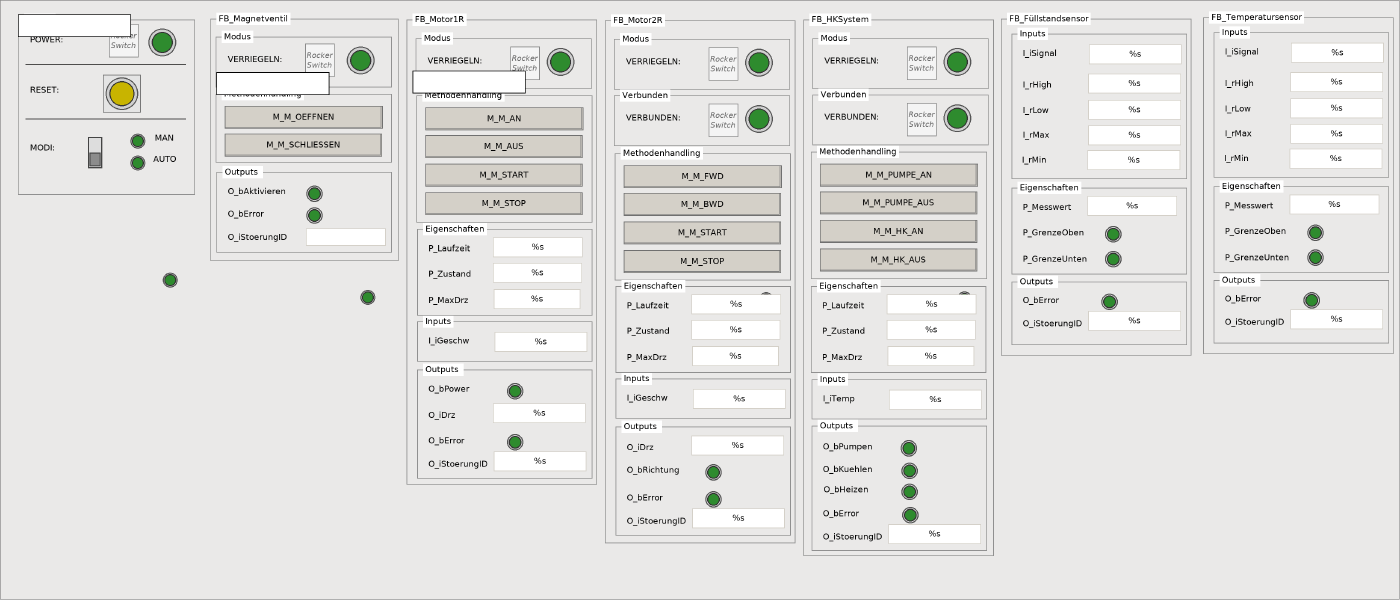
VISUALIZATION Aktoren  // 1863x799
    Rectangle (-1,-1 1863x799)
    GroupBox (280,17 250x330), "FB_Magnetventil"
        Textfield (127,287 106x23), text variable: Reaktoranlage.VENTIL.O_iStoerungID
    GroupBox (287,41 234x75), "Modus"
        Label (13,23 150x30), "VERRIEGELN:"
        Lamp1 (172,18 42x43), variable: Reaktoranlage.VENTIL.I_bVerriegeln, style: Lamp-Lamp1-Green
        Lamp1 (191,340 23x30), style: Lamp-Lamp1-Green
    RockerSwitch (406,58 39x44), variable: Reaktoranlage.VENTIL.I_bVerriegeln, behaviour: TOGGLE, style: Switch-RockerSwitch-Gray
    GroupBox (287,117 234x99), "Methodenhandling"
        Rectangle (-530,-100 150x30)
        Button (12,24 210x30), "M_M_OEFFNEN"
            OnMouseClick: execute { Reaktoranlage.VENTIL.M_M_OEFFNEN(); }
        Button (12,61 209x30), "M_M_SCHLIESSEN"
            OnMouseClick: execute { Reaktoranlage.VENTIL.M_M_SCHLIESSEN(); }
    GroupBox (288,221 233x115), "Outputs"
        Label (12,19 150x30), "O_bAktivieren"
        Label (12,49 150x30), "O_bError"
        Label (12,80 150x30), "O_iStoerungID"
        Lamp1 (118,22 25x30), variable: Reaktoranlage.VENTIL.O_bAktivieren, style: Lamp-Lamp1-Green
        Lamp1 (118,51 25x30), variable: Reaktoranlage.VENTIL.O_bStoerung, style: Lamp-Lamp1-Green
    GroupBox (24,18 235x241), "Modus"
        Label (13,20 150x30), "POWER:"
        RockerSwitch (121,14 39x44), variable: Reaktoranlage.Modus.I_bPower, behaviour: TOGGLE, style: Switch-RockerSwitch-Gray
        Label (13,164 150x30), "MODI:"
        DipSwitch (82,161 41x48), variable: Reaktoranlage.Modus.I_bMode, behaviour: TOGGLE, style: Switch-DipSwitch-Gray
        Lamp1 (148,155 23x30), variable: Reaktoranlage.Modus.O_bMAN, style: Lamp-Lamp1-Green
        Lamp1 (148,184 23x30), variable: Reaktoranlage.Modus.O_bAUTO, style: Lamp-Lamp1-Green
        Label (177,179 46x30), "AUTO"
        Lamp1 (191,340 23x30), style: Lamp-Lamp1-Green
        Line (10,67) (223,67)
        Lamp1 (171,17 42x43), variable: Reaktoranlage.Modus.I_bPower, style: Lamp-Lamp1-Green
        Label (179,151 46x30), "MAN"
        Label (13,87 150x30), "RESET:"
        PushSwitch (113,80 50x53), variable: GVL.VIS_SysReset, behaviour: TAP, style: Switch-PushSwitch-Yellow
        Line (10,140) (223,140)
    GroupBox (541,18 253x627), "FB_Motor1R"
        GroupBox (12,25 234x75), "Modus"
            Label (13,23 150x30), "VERRIEGELN:"
            Lamp1 (172,18 42x43), variable: Reaktoranlage.RUEHRER.I_bVerriegeln, style: Lamp-Lamp1-Green
            Lamp1 (191,340 23x30), style: Lamp-Lamp1-Green
            RockerSwitch (126,19 39x44), variable: Reaktoranlage.RUEHRER.I_bVerriegeln, behaviour: TOGGLE, style: Switch-RockerSwitch-Gray
        GroupBox (13,101 234x177), "Methodenhandling"
            Rectangle (-530,-100 150x30)
            Button (12,24 210x30), "M_M_AN"
                OnMouseClick: execute { Reaktoranlage.RUEHRER.M_M_AN(); }
            Button (12,61 209x30), "M_M_AUS"
                OnMouseClick: execute { Reaktoranlage.RUEHRER.M_M_AUS(); }
            Button (12,99 209x30), "M_M_START"
                OnMouseClick: execute { Reaktoranlage.RUEHRER.M_M_START(); }
            Button (12,137 209x30), "M_M_STOP"
                OnMouseClick: execute { Reaktoranlage.RUEHRER.M_M_STOP(); }
        GroupBox (14,402 233x61), "Inputs"
            Label (12,19 150x30), "I_iGeschw"
            Textfield (103,22 123x26), "%s", text variable: Reaktoranlage.RUEHRER.I_iGeschw
                OnMouseClick: write Reaktoranlage.RUEHRER.I_iGeschw via Edit, min 0
        GroupBox (14,279 233x123), "Eigenschaften"
            Label (12,19 150x30), "P_Laufzeit"
            Label (12,88 150x30), "P_MaxDrz"
            Label (12,53 150x30), "P_Zustand"
            Textfield (101,53 118x26), "%s", text variable: Reaktoranlage.RUEHRER.V_Zustand, input disabled if: TRUE
            Textfield (102,88 115x26), "%s", text variable: Reaktoranlage.RUEHRER.V_DrzMax
                OnMouseClick: write Reaktoranlage.RUEHRER.V_DrzMax via Default
            Textfield (101,19 119x26), "%s", text variable: Reaktoranlage.RUEHRER.V_Zeit, input disabled if: TRUE
        GroupBox (14,466 233x153), "Outputs"
            Label (12,19 150x30), "O_bPower"
            Label (12,88 150x30), "O_bError"
            Label (12,119 150x30), "O_iStoerungID"
            Lamp1 (118,22 25x30), variable: Reaktoranlage.RUEHRER.O_bPower, style: Lamp-Lamp1-Green
            Lamp1 (118,90 25x30), variable: Reaktoranlage.RUEHRER.O_bStoerung, style: Lamp-Lamp1-Green
            Textfield (101,53 123x26), "%s", text variable: Reaktoranlage.RUEHRER.O_iDrz, input disabled if: TRUE
            Textfield (102,117 123x26), "%s", text variable: Reaktoranlage.RUEHRER.O_iStoerungID, input disabled if: TRUE
            Label (12,54 150x30), "O_iDrz"
    GroupBox (805,19 253x704), "FB_Motor2R"
        GroupBox (12,25 234x75), "Modus"
            Label (13,23 150x30), "VERRIEGELN:"
            Lamp1 (172,18 42x43), variable: Reaktoranlage.PUMPE.I_bVerriegeln, style: Lamp-Lamp1-Green
            Lamp1 (191,340 23x30), style: Lamp-Lamp1-Green
            RockerSwitch (126,19 39x44), variable: Reaktoranlage.PUMPE.I_bVerriegeln, behaviour: TOGGLE, style: Switch-RockerSwitch-Gray
        GroupBox (13,177 234x177), "Methodenhandling"
            Rectangle (-530,-100 150x30)
            Button (12,24 210x30), "M_M_FWD"
                OnMouseClick: execute { Reaktoranlage.PUMPE.M_M_FWD(); }
            Button (12,61 209x30), "M_M_BWD"
                OnMouseClick: execute { Reaktoranlage.PUMPE.M_M_BWD(); }
            Button (12,99 209x30), "M_M_START"
                OnMouseClick: execute { Reaktoranlage.PUMPE.M_M_START(); }
            Button (12,137 209x30), "M_M_STOP"
                OnMouseClick: execute { Reaktoranlage.PUMPE.M_M_STOP(); }
        GroupBox (14,477 233x61), "Inputs"
            Label (12,19 150x30), "I_iGeschw"
            Textfield (103,22 123x26), "%s", text variable: Reaktoranlage.PUMPE.I_iGeschw
                OnMouseClick: write Reaktoranlage.PUMPE.I_iGeschw via Edit, min 0
        GroupBox (14,354 233x123), "Eigenschaften"
            Label (12,19 150x30), "P_Laufzeit"
            Label (12,88 150x30), "P_MaxDrz"
            Label (12,53 150x30), "P_Zustand"
            Textfield (101,53 118x26), "%s", text variable: Reaktoranlage.PUMPE.V_Zustand, input disabled if: TRUE
            Textfield (102,88 115x26), "%s", text variable: Reaktoranlage.PUMPE.V_DrzMax
                OnMouseClick: write Reaktoranlage.PUMPE.V_DrzMax via Default
            Textfield (101,19 119x26), "%s", text variable: Reaktoranlage.PUMPE.V_Zeit, input disabled if: TRUE
        GroupBox (14,541 233x153), "Outputs"
            Label (12,51 150x30), "O_bRichtung"
            Label (12,88 150x30), "O_bError"
            Label (12,119 150x30), "O_iStoerungID"
            Lamp1 (118,54 25x30), variable: Reaktoranlage.PUMPE.O_bRichtung, style: Lamp-Lamp1-Green
            Lamp1 (118,90 25x30), variable: Reaktoranlage.PUMPE.O_bStoerung, style: Lamp-Lamp1-Green
            Textfield (101,20 123x26), "%s", text variable: Reaktoranlage.PUMPE.O_iDrz, input disabled if: TRUE
            Textfield (102,117 123x26), "%s", text variable: Reaktoranlage.PUMPE.O_iStoerungID, input disabled if: TRUE
            Label (12,21 150x30), "O_iDrz"
        GroupBox (12,100 234x75), "Verbunden"
            Label (13,23 150x30), "VERBUNDEN:"
            Lamp1 (172,18 42x43), variable: Reaktoranlage.PUMPE.I_bVerbunden, style: Lamp-Lamp1-Green
            RockerSwitch (126,19 39x44), variable: Reaktoranlage.PUMPE.I_bVerbunden, behaviour: TOGGLE, style: Switch-RockerSwitch-Gray
    GroupBox (1069,18 253x722), "FB_HKSystem"
        GroupBox (12,25 234x75), "Modus"
            Label (13,23 150x30), "VERRIEGELN:"
            Lamp1 (172,18 42x43), variable: Reaktoranlage.HKSYSTEM.I_bVerriegeln, style: Lamp-Lamp1-Green
            Lamp1 (191,340 23x30), style: Lamp-Lamp1-Green
            RockerSwitch (126,19 39x44), variable: Reaktoranlage.HKSYSTEM.I_bVerriegeln, behaviour: TOGGLE, style: Switch-RockerSwitch-Gray
        GroupBox (12,100 234x75), "Verbunden"
            Label (13,23 150x30), "VERBUNDEN:"
            Lamp1 (172,18 42x43), variable: Reaktoranlage.HKSYSTEM.I_bVerbunden, style: Lamp-Lamp1-Green
            RockerSwitch (126,19 39x44), variable: Reaktoranlage.HKSYSTEM.I_bVerbunden, behaviour: TOGGLE, style: Switch-RockerSwitch-Gray
        GroupBox (10,176 234x177), "Methodenhandling"
            Rectangle (-530,-100 150x30)
            Button (12,24 210x30), "M_M_PUMPE_AN"
                OnMouseClick: execute { Reaktoranlage.HKSYSTEM.M_M_PUMPE_AN(); }
            Button (12,61 209x30), "M_M_PUMPE_AUS"
                OnMouseClick: execute { Reaktoranlage.HKSYSTEM.M_M_PUMPE_AUS(); }
            Button (12,99 209x30), "M_M_HK_AN"
                OnMouseClick: execute { Reaktoranlage.HKSYSTEM.M_M_HK_AN(); }
            Button (12,137 209x30), "M_M_HK_AUS"
                OnMouseClick: execute { Reaktoranlage.HKSYSTEM.M_M_HK_AUS(); }
        GroupBox (11,541 233x174), "Outputs"
            Label (12,51 150x30), "O_bKuehlen"
            Label (12,110 150x30), "O_bError"
            Label (12,141 150x30), "O_iStoerungID"
            Lamp1 (118,53 25x30), variable: Reaktoranlage.HKSYSTEM.O_bKuehlen, style: Lamp-Lamp1-Green
            Lamp1 (119,112 25x30), variable: Reaktoranlage.HKSYSTEM.O_bStoerung, style: Lamp-Lamp1-Green
            Textfield (102,139 123x26), "%s", text variable: Reaktoranlage.HKSYSTEM.O_iStoerungID, input disabled if: TRUE
            Label (12,21 150x30), "O_bPumpen"
            Label (13,78 150x30), "O_bHeizen"
            Lamp1 (118,81 25x30), variable: Reaktoranlage.HKSYSTEM.O_bHeizen, style: Lamp-Lamp1-Green
            Lamp1 (117,23 25x30), variable: Reaktoranlage.HKSYSTEM.O_bPumpen, style: Lamp-Lamp1-Green
        GroupBox (11,479 233x61), "Inputs"
            Label (12,19 150x30), "I_iTemp"
            Textfield (103,22 123x26), "%s", text variable: Reaktoranlage.HKSYSTEM.I_iTemp
                OnMouseClick: write Reaktoranlage.HKSYSTEM.I_iTemp via Edit, min 0
        GroupBox (10,355 233x123), "Eigenschaften"
            Label (12,19 150x30), "P_Laufzeit"
            Label (12,88 150x30), "P_MaxDrz"
            Label (12,53 150x30), "P_Zustand"
            Textfield (101,53 118x26), "%s", text variable: Reaktoranlage.HKSYSTEM.V_Zustand, input disabled if: TRUE
            Textfield (102,88 115x26), "%s", text variable: Reaktoranlage.HKSYSTEM.V_DefTemp
                OnMouseClick: write Reaktoranlage.HKSYSTEM.V_DefTemp via Default
            Textfield (101,19 119x26), "%s", text variable: Reaktoranlage.HKSYSTEM.V_Zeit, input disabled if: TRUE
    GroupBox (1332,17 253x456), "FB_Füllstandsensor"
        GroupBox (14,20 233x201), "Inputs"
            Label (12,19 150x30), "I_iSignal"
            Textfield (103,22 123x26), "%s", text variable: Reaktoranlage.FUELLSEN.I_iSignal
                OnMouseClick: write Reaktoranlage.FUELLSEN.I_iSignal via Edit, min 0
            Label (12,61 150x30), "I_rHigh"
            Label (12,95 150x30), "I_rLow"
            Label (12,128 150x30), "I_rMax"
            Label (11,161 150x30), "I_rMin"
        GroupBox (14,225 233x123), "Eigenschaften"
            Label (12,19 150x30), "P_Messwert"
            Label (12,88 150x30), "P_GrenzeUnten"
            Label (12,53 150x30), "P_GrenzeOben"
            Textfield (101,19 119x26), "%s", text variable: Reaktoranlage.FUELLSEN.Messwert, input disabled if: TRUE
            Lamp1 (123,55 25x30), variable: Reaktoranlage.FUELLSEN.GrenzeOben, style: Lamp-Lamp1-Green
            Lamp1 (123,88 25x30), variable: Reaktoranlage.FUELLSEN.GrenzeUnten, style: Lamp-Lamp1-Green
        GroupBox (14,350 233x92), "Outputs"
            Label (12,18 150x30), "O_bError"
            Label (12,49 150x30), "O_iStoerungID"
            Lamp1 (118,20 25x30), variable: Reaktoranlage.FUELLSEN.O_bStoerung, style: Lamp-Lamp1-Green
            Textfield (102,47 123x26), "%s", text variable: Reaktoranlage.PUMPE.O_iStoerungID, input disabled if: TRUE
        Textfield (116,81 123x26), "%s", text variable: Reaktoranlage.FUELLSEN.I_rHigh
            OnMouseClick: write Reaktoranlage.FUELLSEN.I_rHigh via Edit, min 0
        Textfield (116,116 123x26), "%s", text variable: Reaktoranlage.FUELLSEN.I_rMin
            OnMouseClick: write Reaktoranlage.FUELLSEN.I_rLow via Edit, min 0
        Textfield (116,150 123x26), "%s", text variable: Reaktoranlage.FUELLSEN.I_rMax
            OnMouseClick: write Reaktoranlage.FUELLSEN.I_rMax via Edit, min 0
        Textfield (115,183 123x26), "%s", text variable: Reaktoranlage.FUELLSEN.I_rMin
            OnMouseClick: write Reaktoranlage.FUELLSEN.I_rMin via Edit, min 0
    GroupBox (1601,15 253x456), "FB_Temperatursensor"
        GroupBox (14,20 233x201), "Inputs"
            Label (12,19 150x30), "I_iSignal"
            Textfield (103,22 123x26), "%s", text variable: Reaktoranlage.FUELLSEN.I_iSignal
                OnMouseClick: write Reaktoranlage.TEMPSEN.I_rMin via Edit, min 0
            Label (12,61 150x30), "I_rHigh"
            Label (12,95 150x30), "I_rLow"
            Label (12,128 150x30), "I_rMax"
            Label (11,161 150x30), "I_rMin"
        GroupBox (14,225 233x123), "Eigenschaften"
            Label (12,19 150x30), "P_Messwert"
            Label (12,88 150x30), "P_GrenzeUnten"
            Label (12,53 150x30), "P_GrenzeOben"
            Textfield (101,19 119x26), "%s", text variable: Reaktoranlage.TEMPSEN.Messwert, input disabled if: TRUE
            Lamp1 (123,55 25x30), variable: Reaktoranlage.TEMPSEN.GrenzeOben, style: Lamp-Lamp1-Green
            Lamp1 (123,88 25x30), variable: Reaktoranlage.TEMPSEN.GrenzeUnten, style: Lamp-Lamp1-Green
        GroupBox (14,350 233x92), "Outputs"
            Label (12,18 150x30), "O_bError"
            Label (12,49 150x30), "O_iStoerungID"
            Lamp1 (118,20 25x30), variable: Reaktoranlage.TEMPSEN.O_bStoerung, style: Lamp-Lamp1-Green
            Textfield (102,47 123x26), "%s", text variable: Reaktoranlage.TEMPSEN.O_iStoerungID, input disabled if: TRUE
        Textfield (116,81 123x26), "%s", text variable: Reaktoranlage.FUELLSEN.I_rHigh
            OnMouseClick: write Reaktoranlage.TEMPSEN.I_rHigh via Edit, min 0
        Textfield (116,116 123x26), "%s", text variable: Reaktoranlage.FUELLSEN.I_rMin
            OnMouseClick: write Reaktoranlage.TEMPSEN.I_rLow via Edit, min 0
        Textfield (116,150 123x26), "%s", text variable: Reaktoranlage.FUELLSEN.I_rMax
            OnMouseClick: write Reaktoranlage.TEMPSEN.I_rMax via Edit, min 0
        Textfield (115,183 123x26), "%s", text variable: Reaktoranlage.TEMPSEN.O_iStoerungID
            OnMouseClick: write Reaktoranlage.TEMPSEN.I_rMin via Edit, min 0
END_VISUALIZATION

(* stored: Version 1.1.0.1, ProductVersion 3.1.4024.12
   Visu Aktoren: Id {ac277a63-1cee-4a87-a068-9fd3f4af00ac} *)
